// TwinCAT 3 PLC project leader_main
// ProgramVersion: 3.1.4020.4
// libraries:
//   LCLS Motion Control, * (SLAC)
//   Tc2_MC2, * (Beckhoff Automation GmbH)
//   Tc2_Standard, * (Beckhoff Automation GmbH)
//   Tc2_System, * (Beckhoff Automation GmbH)
//   Tc3_Module, * (Beckhoff Automation GmbH)
// project tree:
//   DUTs/ ST_BeamDemand.TcDUT, ST_BisscEncoder.TcDUT, ST_Stepper.TcDUT
//   GVLs/ StepperGVLs.TcGVL
//   / PlcTask.TcTTO
//   POUs/ count_mgr_test.TcPOU, FB_MotorRepeater.TcPOU (not stored), FB_StepperWrapper.TcPOU (not stored), FUN_BisscEvaluator.TcPOU, MAIN.TcPOU
// real-time tasks:
//   TASK PlcTask: cycle T#10ms, priority 20, ADS port 350
// motion (NC):
//   TASK NC-Task 1 SAF: cycle T#2ms, priority 4, ADS port 501
//   TASK NC-Task 1 SVB: cycle T#10ms, priority 8, ADS port 511
//   AXIS Axis 2 (id 2)
//     Velo: RefSearch=1, RefSync=1, SlowManual=1, FastManual=1, Maximum=1
//     OtherSettings: AllowMotionCmdToSlave=true, PulseDistancePos=1, PulseDistanceNeg=1
//     encoder EncType=29
//       EncPara: ScaleFactorNumerator=5e-005, MaxCount=#xffffffff
//         SoftEndMinControl: Enable=true, Range=23
//         SoftEndMaxControl: Enable=true, Range=55
//         Inc: RefSoftSyncMask=#x0000ffff
//     drive DrvType=24
//       Analog: VeloReferenz=25.4
//       TimeComp: TaskDelayCycles=1
//     controller CtrType=1
//       CtrPara: PriorControlFactor=1
//         Observer: BandWidth=20
// I/O:
//   DEVICE Device 1 (EtherCAT), AmsNetId 5.45.6.154.2.1
//     Term 1 (EK1200) [EK1200-5000 EtherCAT Power supply (2A E-Bus)]
//       Term 2 (EL7041) [EL7041 1Ch. Stepper motor output stage (50V, 5A)]
//       Term 3 (EL5042) [EL5042 2Ch. BiSS-C Encoder]
//       Term 4 (EL6695) [EL6695 EtherCAT Bridge terminal (Primary)]
//       Term 5 (EL2124) [EL2124 4Ch. Dig. Output 5V, 20mA]
//       Term 6 (EL9011) [EL9011 End Terminal]
//   DEVICE Device 4 (EtherCAT) (disabled), AmsNetId 5.45.6.154.5.1
//     Box 7 (P00030924 R00010420) [P00030924 R00010420]
//   DEVICE Device 3 (USB) (disabled)
//     Box 1 (CX2100 Power Supply)
//   DEVICE Device 5 (NOV-DP-RAM) (disabled)
// variable links:
//   NC-Task 1 SAF/Axes/Axis 2 <-> Device 1 (EtherCAT)/Term 1 (EK1200)/Term 2 (EL7041)
//     Drive/Inputs/In/nState1 @bit 3 <-> STM Status/Status/Error
//     Drive/Inputs/In/nState1 @bit 5 <-> STM Status/Status/Moving negative
//     Drive/Inputs/In/nState1 @bit 4 <-> STM Status/Status/Moving positive
//     Drive/Inputs/In/nState1 @bit 1 <-> STM Status/Status/Ready
//     Drive/Inputs/In/nState1 <-> STM Status/Status/Ready to enable
//     Drive/Inputs/In/nState1 @bit 6 <-> STM Status/Status/Torque reduced
//     Drive/Inputs/In/nState1 @bit 2 <-> STM Status/Status/Warning
//     Drive/Inputs/In/nState2 @bit 3 <-> STM Status/Status/Digital input 1
//     Drive/Inputs/In/nState2 @bit 4 <-> STM Status/Status/Digital input 2
//     Drive/Inputs/In/nState4 @bit 1 <-> WcState/InputToggle
//     Drive/Inputs/In/nState4 <-> WcState/WcState
//     Drive/Outputs/Out/nCtrl1 <-> STM Control/Control/Enable
//     Drive/Outputs/Out/nCtrl1 @bit 2 <-> STM Control/Control/Reduce torque
//     Drive/Outputs/Out/nCtrl1 @bit 1 <-> STM Control/Control/Reset
//     Drive/Outputs/Out/nDataOut2[0] <-> STM Velocity/Velocity
//   NC-Task 1 SAF/Axes/Axis 2 <-> Device 1 (EtherCAT)/Term 1 (EK1200)/Term 3 (EL5042)
//     Enc/Inputs/In/nComState @bit 1 <-> WcState/InputToggle
//     Enc/Inputs/In/nComState <-> WcState/WcState
//     Enc/Inputs/In/nDataIn1 <-> FB Inputs Channel 1/Position
//     Enc/Inputs/In/nState1 @bit 12 <-> FB Inputs Channel 1/Status/Diag
//     Enc/Inputs/In/nState1 @bit 1 <-> FB Inputs Channel 1/Status/Error
//     Enc/Inputs/In/nState1 @bit 14 <-> FB Inputs Channel 1/Status/Input cycle counter
//     Enc/Inputs/In/nState1 @bit 2 <-> FB Inputs Channel 1/Status/Ready
//     Enc/Inputs/In/nState1 @bit 13 <-> FB Inputs Channel 1/Status/TxPDO State
//     Enc/Inputs/In/nState1 <-> FB Inputs Channel 1/Status/Warning
//   leader_main Instance <-> Device 1 (EtherCAT)/Term 1 (EK1200)/Term 3 (EL5042)
//     PlcTask Inputs/MAIN.Encoder0.encLoc <-> FB Inputs Channel 1/Position
//   leader_main Instance <-> NC-Task 1 SAF/Axes/Axis 2
//     PlcTask Inputs/MAIN.Stepper0.Axis.NcToPlc <-> Outputs/ToPlc
//     PlcTask Outputs/MAIN.Stepper0.Axis.PlcToNc <-> Inputs/FromPlc

CONFIGURATION leader_main
    RESOURCE PLC ON TwinCAT3
        TASK PlcTask(INTERVAL := T#10ms, PRIORITY := 20);
        PROGRAM MAIN WITH PlcTask : MAIN;
    END_RESOURCE
END_CONFIGURATION

// ---- DUTs/ST_BeamDemand.TcDUT
TYPE ST_BeamDemand :
STRUCT
	// What beam rate is required from a device? (Probably units of frequency) 
	beamRate : LREAL;
	// Demand specifies if this demand is an emergency (True). Non-Demand is for non-emergencies
	demand : BOOL;
END_STRUCT
END_TYPE

// ---- DUTs/ST_BisscEncoder.TcDUT
TYPE ST_BisscEncoder :
STRUCT
	// Inclusive limits on encoder position (checks for values exceeding this inclusive range)
	// These values are just guesses - no units yet - no actual data - CHANGE BEFORE USE
	ncLLimit :	ULINT := 0;
	ncULimit :	ULINT := 100;
	// Readback for linear encoder's position
	encLoc	AT %I*	:	ULINT;
END_STRUCT
END_TYPE

// ---- DUTs/ST_Stepper.TcDUT
TYPE ST_Stepper :
STRUCT
	Axis	:	AXIS_REF;
	llimit	:	ULINT	:=	460000;
	ulimit	:	ULINT	:=	1099600;
END_STRUCT
END_TYPE

// ---- GVLs/StepperGVLs.TcGVL
{attribute 'qualified_only'}
VAR_GLOBAL
END_VAR

// ---- POUs/MAIN.TcPOU
PROGRAM MAIN
VAR
	Counter0Inc : DWORD := 1;
	Counter0Read : DWORD; 
	Counter0 : count_mgr_test;
	//Encoder0Read : ULINT;
	Encoder0	:	ST_BisscEncoder;
	EncoderDemand0 : ST_BeamDemand;
	Stepper0	:	ST_Stepper;
	Stepper0EnbP	:	BOOL;
	Stepper0EnbN	:	BOOL;
	
	StepperAxis	:	ST_BasicAxis;
	StepperControl	:	FB_BasicAxisControl;
	StepperMode	:	E_AxisMoveMode;
	StepperState	:	E_AxisMotionState;
	
	fbPower	:	MC_Power;
	//fbJog	:	MC_Jog;
	fbHome	:	MC_Home;
	//fbReadStatus	:	MC_ReadStatus;
	
	fbMoveAbsolute	:	MC_MoveAbsolute;
	fbMoveRelative	:	MC_MoveRelative;
	
END_VAR

//set constants
Encoder0.ncULimit := 170;

//runtime
Counter0(Increment:=Counter0Inc);
Counter0Read := Counter0.CurrentOut;
EncoderDemand0 := FUN_BisscEvaluator(Encoder0);


StepperAxis.stAxis := Stepper0.Axis;
StepperAxis.wMode := StepperMode;
StepperAxis.eState := StepperState;




(*
Stepper0EnbP := Encoder0.encLoc < Stepper0.ulimit;
Stepper0EnbN := Encoder0.encLoc > Stepper0.llimit;

fbPower(Axis:=Stepper0.Axis,Enable:=TRUE,Enable_Positive:=Stepper0EnbP,Enable_Negative:=Stepper0EnbN,Override:=100);
IF fbPower.Status THEN
	fbMoveAbsolute(Axis:=Stepper0.Axis,Velocity:=1);
END_IF

*)

END_PROGRAM

// ---- POUs/count_mgr_test.TcPOU
FUNCTION_BLOCK count_mgr_test
VAR_INPUT
	Increment : DWORD;
END_VAR
VAR_OUTPUT
	CurrentOut : DWORD;
END_VAR
VAR
	UpperLimit : DWORD := 500;
END_VAR
VAR PERSISTENT
	CurrentVal : DWORD := 0;
END_VAR

IF CurrentVal >= UpperLimit THEN
	CurrentVal := 0;
ELSE
	CurrentVal := CurrentVal + Increment;
END_IF



CurrentOut := CurrentVal;

END_FUNCTION_BLOCK

// ---- POUs/FUN_BisscEvaluator.TcPOU
FUNCTION FUN_BisscEvaluator : ST_BeamDemand
VAR_INPUT
	encoder : ST_BisscEncoder;
END_VAR
VAR	
	readLoc: ULINT;
	newDemand : ST_BeamDemand;
END_VAR

readLoc := Encoder.encLoc;
IF readLoc <= Encoder.ncULimit THEN
	newDemand.demand := TRUE;
ELSE
	newDemand.demand := FALSE;
END_IF

IF readLoc <= Encoder.ncULimit THEN 
	newDemand.beamRate := 0;
ELSE
	newDemand.beamRate := 50;
END_IF

FUN_BisscEvaluator := newDemand;

END_FUNCTION
